FUNCTION_BLOCK WRITE_VIDEO2FILE (* Template for a Basic Function Block Type *)
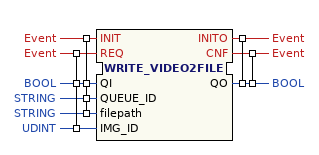
  EVENT_INPUT
    INIT WITH QI, filepath, QUEUE_ID; (* Initialization Request *)
    REQ WITH QI, IMG_ID; (* Normal Execution Request *)
  END_EVENT
  EVENT_OUTPUT
    INITO WITH QO; (* Initialization Confirm *)
    CNF WITH QO; (* Execution Confirmation *)
  END_EVENT
  VAR_INPUT
    QI : BOOL; (* Input event qualifier *)
    QUEUE_ID : STRING;
    filepath : STRING;
    IMG_ID : UDINT;
  END_VAR
  VAR_OUTPUT
    QO : BOOL; (* Output event qualifier *)
  END_VAR
END_FUNCTION_BLOCK
